(* IEC 61131-3 sources: cc_kush_rewrite/Dumper/POU/Hardware, 4 files *)

(* ---- FB_DumperConveyorMotors.st ---- *)
FUNCTION_BLOCK FB_DumperConveyorMotors
VAR_INPUT
	Dumper : REFERENCE TO ST_Dumper;
	xStart : BOOL;              // Команда запуска
	xStop : BOOL;               // Команда остановки
	xEmergencyStop : BOOL;      // Аварийная остановка
	rTargetFrequency : REAL;    // Целевая частота моторов
END_VAR
VAR_OUTPUT
	eStage : E_StageActuator;   // Текущая стадия
	rCurrentFrequency : REAL;   // Текущая частота моторов (среднее значение)
END_VAR
VAR
	STAGE : E_StageActuator := E_StageActuator.IDLE;

	// Подстадии запуска
	nStartingSubstage : INT := 0;
	// 0 - RELEASE_BRAKE: Отпускание тормоза
	// 1 - WAIT_BRAKE_FEEDBACK: Ожидание обратной связи тормоза
	// 2 - START_VFD: Запуск VFD

	// Подстадии остановки
	nStoppingSubstage : INT := 0;
	// 0 - Нормальная работа
	// 1 - STOP_VFD: Остановка VFD
	// 2 - WAIT_VFD_STOP: Ожидание остановки VFD
	// 3 - ACTIVATE_BRAKE: Активация тормоза
	// 4 - WAIT_BRAKE_FEEDBACK: Ожидание обратной связи тормоза

	// Таймер задержки включения тормоза
	tonTimerEnableBrake : TON;

	// Флаг запуска таймера (защита от зацикливания)
	xBrakeTimerStarted : BOOL := FALSE;
END_VAR

// ========================================
// FB_DumperConveyorMotors - Управление моторами конвейера отвалообразователя
// ========================================
//
// НАЗНАЧЕНИЕ:
// - Управление двумя моторами конвейера (22 кВт каждый)
// - Прямой пуск (без плавного разгона)
// - Последовательная остановка (VFD → тормоз)
// - Не знает про ППЗ и верхнеуровневую логику
// - Просто выполняет команды START/STOP
//
// ВХОДЫ:
// - xStart: команда запуска моторов
// - xStop: команда остановки моторов
// - xEmergencyStop: аварийная остановка
// - rTargetFrequency: целевая частота (Гц)
//
// ВЫХОДЫ:
// - eStage: текущая стадия (IDLE/STARTING/WORK)
// - rCurrentFrequency: текущая частота моторов
//
// ========================================

// ========================================
// ПРИОРИТЕТНАЯ ОБРАБОТКА АВАРИЙНОЙ ОСТАНОВКИ
// ========================================

IF xEmergencyStop THEN
	// Аварийная остановка: немедленное выключение VFD
	Dumper.MotorConveyor[1].VFD.qxStart := FALSE;
	Dumper.MotorConveyor[2].VFD.qxStart := FALSE;

	// Активация тормоза
	Dumper.qxBreakerConveyor := FALSE;

	// Переход в IDLE
	STAGE := E_StageActuator.IDLE;
	nStartingSubstage := 0;
	nStoppingSubstage := 0;
	tonTimerEnableBrake(IN := FALSE);
	xBrakeTimerStarted := FALSE;
END_IF

// ========================================
// АВТОМАТ УПРАВЛЕНИЯ МОТОРАМИ
// ========================================

CASE STAGE OF
	E_StageActuator.IDLE:
		// Сброс подстадий
		nStartingSubstage := 0;
		nStoppingSubstage := 0;

		// Сброс флага таймера тормоза
		xBrakeTimerStarted := FALSE;

		// Тормоз активен (удерживает механизм)
		Dumper.qxBreakerConveyor := FALSE;

		// Команда запуска
		IF xStart AND NOT xEmergencyStop THEN
			STAGE := E_StageActuator.STARTING;
		END_IF

	E_StageActuator.STARTING:
		// Проверка команды остановки во время запуска
		IF xStop THEN
			// Прервать запуск и перейти к остановке
			STAGE := E_StageActuator.WORK;
			nStartingSubstage := 0;
			nStoppingSubstage := 1; // Начать процедуру остановки
		END_IF

		// Последовательный запуск: Тормоз → VFD → Разгон
		CASE nStartingSubstage OF
			0: // RELEASE_BRAKE - Отпускание тормоза
				// Отпустить тормоз (1 = тормоз отпущен)
				Dumper.qxBreakerConveyor := TRUE;

				// Переход к следующей подстадии
				nStartingSubstage := 1;

			1: // WAIT_BRAKE_FEEDBACK - Ожидание обратной связи тормоза
				// Получить обратную связь реле тормоза
				IF Dumper.fbBreakerConveyor.qxSignal THEN
					// Обратная связь получена, переходим к запуску VFD
					nStartingSubstage := 2;
				END_IF

			2: // START_VFD - Запуск VFD
				// Команда ПУСК на частотный преобразователь
				Dumper.MotorConveyor[1].VFD.qxStart := TRUE;
				Dumper.MotorConveyor[2].VFD.qxStart := TRUE;

				// Если оба VFD запущены (обратная связь)
				IF Dumper.MotorConveyor[1].VFD.fbStateIsWorking.qxSignal
					AND Dumper.MotorConveyor[2].VFD.fbStateIsWorking.qxSignal
				THEN
					// Переход в режим WORK
					STAGE := E_StageActuator.WORK;
					nStartingSubstage := 0;
				END_IF
		END_CASE;

	E_StageActuator.WORK:
		// Нормальная работа или штатная остановка через подстадии
		CASE nStoppingSubstage OF
			0: // Нормальная работа
				// Команда остановки
				IF xStop THEN
					nStoppingSubstage := 1;
				END_IF

			1: // STOP_VFD - Остановка VFD
				// Отключить команду пуска на VFD
				Dumper.MotorConveyor[1].VFD.qxStart := FALSE;
				Dumper.MotorConveyor[2].VFD.qxStart := FALSE;

				nStoppingSubstage := 2;

			2: // WAIT_VFD_STOP - Ожидание остановки VFD
				// Проверить обратную связь VFD о выключении
				IF NOT Dumper.MotorConveyor[1].VFD.fbStateIsWorking.qxSignal
					AND NOT Dumper.MotorConveyor[2].VFD.fbStateIsWorking.qxSignal
				THEN
					nStoppingSubstage := 3;
				END_IF

			3: // ACTIVATE_BRAKE - Активация тормоза с задержкой
				// Включение таймера на задержку тормоза (один раз)
				IF NOT xBrakeTimerStarted THEN
					xBrakeTimerStarted := TRUE;
				END_IF

				tonTimerEnableBrake(IN := xBrakeTimerStarted, PT := T#5S);

				IF tonTimerEnableBrake.Q THEN
					// Снять сигнал с тормоза (FALSE = активен)
					Dumper.qxBreakerConveyor := FALSE;
					tonTimerEnableBrake(IN := FALSE);
					xBrakeTimerStarted := FALSE;
					nStoppingSubstage := 4;
				END_IF

			4: // WAIT_BRAKE_FEEDBACK - Переход в IDLE
				STAGE := E_StageActuator.IDLE;
				nStoppingSubstage := 0;
		END_CASE;
END_CASE;

// ========================================
// ЗАДАНИЕ ЧАСТОТЫ МОТОРОВ
// ========================================

// Установка частоты напрямую в аналоговый выход VFD
// В режиме IDLE и при остановке частота = 0
// В режиме WORK частота = rTargetFrequency
IF STAGE = E_StageActuator.WORK THEN
	Dumper.MotorConveyor[1].VFD.qrOutFrequency := rTargetFrequency;
	Dumper.MotorConveyor[2].VFD.qrOutFrequency := rTargetFrequency;
ELSE
	Dumper.MotorConveyor[1].VFD.qrOutFrequency := 0.0;
	Dumper.MotorConveyor[2].VFD.qrOutFrequency := 0.0;
END_IF;

// ========================================
// ВЫХОДЫ
// ========================================

// Текущая стадия
eStage := STAGE;

// Текущая частота (среднее значение двух моторов)
rCurrentFrequency := (Dumper.MotorConveyor[1].VFD.rActualFrequency
                    + Dumper.MotorConveyor[2].VFD.rActualFrequency) / 2.0;

END_FUNCTION_BLOCK

(* ---- FB_DumperMotorErrors.st ---- *)
FUNCTION_BLOCK FB_DumperMotorErrors
VAR_INPUT
	Dumper : REFERENCE TO ST_Dumper;
END_VAR
VAR_OUTPUT
	// Ошибки моторов конвейера
	xErrorMotorConv1 : BOOL;
	xErrorMotorConv2 : BOOL;
	xErrorMotorConv_Any : BOOL;

	// Ошибки моторов поворота
	xErrorMotorRot1 : BOOL;
	xErrorMotorRot2 : BOOL;
	xErrorMotorRot_Any : BOOL;

	// Агрегированный выход
	xErrorMotors : BOOL; // Любая ошибка моторов
END_VAR

// ========================================
// FB_DumperMotorErrors - Проверка ошибок моторов отвалообразователя
// ========================================
//
// НАЗНАЧЕНИЕ:
// - Проверка всех моторов отвалообразователя на ошибки
// - Формирование индивидуальных флагов ошибок
// - Агрегирование ошибок
//
// МОТОРЫ:
// - MotorConveyor[1..2]: Моторы конвейера (22 кВт)
// - MotorRotation[1..2]: Моторы поворота (3 кВт)
//
// ПРОВЕРЯЕМЫЕ ОШИБКИ:
// - Ошибка VFD (fbStateFailure: 0 = ошибка, 1 = норма, NC контакт)
//
// ========================================

// ========================================
// ПРОВЕРКА МОТОРОВ КОНВЕЙЕРА
// ========================================

// Мотор конвейера 1
// fbStateFailure - NC контакт: 0 = ошибка VFD, 1 = норма
xErrorMotorConv1 := NOT Dumper.MotorConveyor[1].VFD.fbStateFailure.qxSignal;

// Мотор конвейера 2
xErrorMotorConv2 := NOT Dumper.MotorConveyor[2].VFD.fbStateFailure.qxSignal;

xErrorMotorConv_Any := xErrorMotorConv1 OR xErrorMotorConv2;

// ========================================
// ПРОВЕРКА МОТОРОВ ПОВОРОТА
// ========================================

// Мотор поворота 1
xErrorMotorRot1 := NOT Dumper.MotorRotation[1].VFD.fbStateFailure.qxSignal;

// Мотор поворота 2
xErrorMotorRot2 := NOT Dumper.MotorRotation[2].VFD.fbStateFailure.qxSignal;

xErrorMotorRot_Any := xErrorMotorRot1 OR xErrorMotorRot2;

// ========================================
// АГРЕГИРОВАНИЕ ОШИБОК
// ========================================

xErrorMotors := xErrorMotorConv_Any OR xErrorMotorRot_Any;

END_FUNCTION_BLOCK

(* ---- FB_DumperRotationMotors.st ---- *)
FUNCTION_BLOCK FB_DumperRotationMotors
VAR_INPUT
	Dumper : REFERENCE TO ST_Dumper;
	xTurnLeft : BOOL;           // Команда поворота влево
	xTurnRight : BOOL;          // Команда поворота вправо
	xStop : BOOL;               // Команда остановки поворота
	xEmergencyStop : BOOL;      // Аварийная остановка
	rTargetFrequency : REAL;    // Целевая частота моторов
END_VAR
VAR_OUTPUT
	eStage : E_StageActuator;   // Текущая стадия
	rCurrentFrequency : REAL;   // Текущая частота моторов (среднее значение)
	xRotatingLeft : BOOL;       // Активен поворот влево
	xRotatingRight : BOOL;      // Активен поворот вправо
END_VAR
VAR
	STAGE : E_StageActuator := E_StageActuator.IDLE;

	// Направление поворота
	xLeftActive : BOOL := FALSE;  // Поворот влево активен
	xRightActive : BOOL := FALSE; // Поворот вправо активен

	// Подстадии запуска
	nStartingSubstage : INT := 0;
	// 0 - IDLE
	// 1 - RELEASE_BRAKE: Отпускание тормоза поворота
	// 2 - WAIT_BRAKE_FEEDBACK: Ожидание обратной связи тормоза
	// 3 - START_VFD: Запуск VFD поворота

	// Подстадии остановки
	nStoppingSubstage : INT := 0;
	// 0 - Нормальная работа
	// 1 - STOP_VFD: Остановка VFD
	// 2 - WAIT_VFD_STOP: Ожидание остановки VFD
	// 3 - ACTIVATE_BRAKE: Активация тормоза

	// Таймер задержки включения тормоза
	tonTimerEnableBrake : TON;

	// Флаг запуска таймера (защита от зацикливания)
	xBrakeTimerStarted : BOOL := FALSE;
END_VAR

// ========================================
// FB_DumperRotationMotors - Управление моторами поворота отвалообразователя
// ========================================
//
// НАЗНАЧЕНИЕ:
// - Управление двумя моторами поворота (3 кВт каждый)
// - Поддержка реверса (влево/вправо)
// - Блокировка по концевым выключателям
// - Последовательная остановка (VFD → тормоз)
// - Не знает про верхнеуровневую логику
// - Просто выполняет команды TURN_LEFT/TURN_RIGHT/STOP
//
// ВХОДЫ:
// - xTurnLeft: команда поворота влево
// - xTurnRight: команда поворота вправо
// - xStop: команда остановки
// - xEmergencyStop: аварийная остановка
// - rTargetFrequency: целевая частота (Гц)
//
// ВЫХОДЫ:
// - eStage: текущая стадия (IDLE/STARTING/WORK)
// - rCurrentFrequency: текущая частота моторов
// - xRotatingLeft: флаг активного поворота влево
// - xRotatingRight: флаг активного поворота вправо
//
// ========================================

// ========================================
// ПРИОРИТЕТНАЯ ОБРАБОТКА АВАРИЙНОЙ ОСТАНОВКИ
// ========================================

IF xEmergencyStop THEN
	// Аварийная остановка: немедленное выключение VFD
	Dumper.MotorRotation[1].VFD.qxStart := FALSE;
	Dumper.MotorRotation[2].VFD.qxStart := FALSE;
	Dumper.MotorRotation[1].qxVFDReverseStart := FALSE;
	Dumper.MotorRotation[2].qxVFDReverseStart := FALSE;

	// Активация тормоза
	Dumper.qxBreakerRotation := FALSE;

	// Сброс направления
	xLeftActive := FALSE;
	xRightActive := FALSE;

	// Переход в IDLE
	STAGE := E_StageActuator.IDLE;
	nStartingSubstage := 0;
	nStoppingSubstage := 0;
	tonTimerEnableBrake(IN := FALSE);
	xBrakeTimerStarted := FALSE;
END_IF

// ========================================
// АВТОМАТ УПРАВЛЕНИЯ МОТОРАМИ ПОВОРОТА
// ========================================

CASE STAGE OF
	E_StageActuator.IDLE:
		// Сброс подстадий
		nStartingSubstage := 0;
		nStoppingSubstage := 0;

		// Сброс флага таймера тормоза
		xBrakeTimerStarted := FALSE;

		// Тормоз активен
		Dumper.qxBreakerRotation := FALSE;

		// Остановка VFD
		Dumper.MotorRotation[1].VFD.qxStart := FALSE;
		Dumper.MotorRotation[2].VFD.qxStart := FALSE;
		Dumper.MotorRotation[1].qxVFDReverseStart := FALSE;
		Dumper.MotorRotation[2].qxVFDReverseStart := FALSE;

		// Сброс флагов направления
		xLeftActive := FALSE;
		xRightActive := FALSE;

		// Команда поворота влево
		IF xTurnLeft AND NOT xEmergencyStop AND NOT xTurnRight THEN
			// Проверка концевого выключателя влево
			// qxSignal = TRUE означает концевик в норме (не нажат)
			IF Dumper.fbEndSwitchLeft.qxSignal THEN
				xLeftActive := TRUE;
				xRightActive := FALSE;
				STAGE := E_StageActuator.STARTING;
			END_IF
		END_IF

		// Команда поворота вправо
		IF xTurnRight AND NOT xEmergencyStop AND NOT xTurnLeft THEN
			// Проверка концевого выключателя вправо
			IF Dumper.fbEndSwitchRight.qxSignal THEN
				xRightActive := TRUE;
				xLeftActive := FALSE;
				STAGE := E_StageActuator.STARTING;
			END_IF
		END_IF

	E_StageActuator.STARTING:
		// Проверка команды остановки во время запуска
		IF xStop THEN
			// Прервать запуск и перейти к остановке
			STAGE := E_StageActuator.WORK;
			nStartingSubstage := 0;
			nStoppingSubstage := 1; // Начать процедуру остановки
		END_IF

		// Проверка достижения концевого выключателя
		IF (xLeftActive AND NOT Dumper.fbEndSwitchLeft.qxSignal)
			OR (xRightActive AND NOT Dumper.fbEndSwitchRight.qxSignal)
		THEN
			// Концевик достигнут, начать остановку
			STAGE := E_StageActuator.WORK;
			nStartingSubstage := 0;
			nStoppingSubstage := 1;
		END_IF

		// Последовательный запуск: Тормоз → VFD → Разгон
		CASE nStartingSubstage OF
			0: // IDLE
				nStartingSubstage := 1;

			1: // RELEASE_BRAKE - Отпускание тормоза
				// Отпустить тормоз (1 = тормоз отпущен)
				Dumper.qxBreakerRotation := TRUE;

				// Переход к следующей подстадии
				nStartingSubstage := 2;

			2: // WAIT_BRAKE_FEEDBACK - Ожидание обратной связи тормоза
				// Получить обратную связь реле тормоза
				IF Dumper.fbBreakerRotation.qxSignal THEN
					// Обратная связь получена, переходим к запуску VFD
					nStartingSubstage := 3;
				END_IF

			3: // START_VFD - Запуск VFD
				// Установка направления и запуск VFD
				IF xLeftActive THEN
					// Поворот влево - прямое направление
					Dumper.MotorRotation[1].qxVFDReverseStart := FALSE;
					Dumper.MotorRotation[2].qxVFDReverseStart := FALSE;
					Dumper.MotorRotation[1].VFD.qxStart := TRUE;
					Dumper.MotorRotation[2].VFD.qxStart := TRUE;
				ELSIF xRightActive THEN
					// Поворот вправо - реверс
					Dumper.MotorRotation[1].VFD.qxStart := FALSE;
					Dumper.MotorRotation[2].VFD.qxStart := FALSE;
					Dumper.MotorRotation[1].qxVFDReverseStart := TRUE;
					Dumper.MotorRotation[2].qxVFDReverseStart := TRUE;
				END_IF

				// Проверка запуска VFD (обратная связь)
				IF Dumper.MotorRotation[1].VFD.fbStateIsWorking.qxSignal
					AND Dumper.MotorRotation[2].VFD.fbStateIsWorking.qxSignal
				THEN
					// VFD запущены, переходим в режим работы
					STAGE := E_StageActuator.WORK;
					nStartingSubstage := 0;
				END_IF
		END_CASE;

	E_StageActuator.WORK:
		// Нормальная работа или штатная остановка через подстадии
		CASE nStoppingSubstage OF
			0: // Нормальная работа
				// Проверка команды остановки
				IF xStop THEN
					nStoppingSubstage := 1;
				END_IF

				// Проверка достижения концевого выключателя
				IF (xLeftActive AND NOT Dumper.fbEndSwitchLeft.qxSignal)
					OR (xRightActive AND NOT Dumper.fbEndSwitchRight.qxSignal)
				THEN
					// Концевик достигнут, автоматическая остановка
					nStoppingSubstage := 1;
				END_IF

			1: // STOP_VFD - Остановка VFD
				// Отключить команду пуска на VFD
				Dumper.MotorRotation[1].VFD.qxStart := FALSE;
				Dumper.MotorRotation[2].VFD.qxStart := FALSE;
				Dumper.MotorRotation[1].qxVFDReverseStart := FALSE;
				Dumper.MotorRotation[2].qxVFDReverseStart := FALSE;

				nStoppingSubstage := 2;

			2: // WAIT_VFD_STOP - Ожидание остановки VFD
				// Проверить обратную связь VFD о выключении
				IF NOT Dumper.MotorRotation[1].VFD.fbStateIsWorking.qxSignal
					AND NOT Dumper.MotorRotation[2].VFD.fbStateIsWorking.qxSignal
				THEN
					nStoppingSubstage := 3;
				END_IF

			3: // ACTIVATE_BRAKE - Активация тормоза с задержкой
				// Включение таймера на задержку тормоза (один раз)
				IF NOT xBrakeTimerStarted THEN
					xBrakeTimerStarted := TRUE;
				END_IF

				tonTimerEnableBrake(IN := xBrakeTimerStarted, PT := T#3S);

				IF tonTimerEnableBrake.Q THEN
					// Снять сигнал с тормоза (FALSE = активен)
					Dumper.qxBreakerRotation := FALSE;
					tonTimerEnableBrake(IN := FALSE);
					xBrakeTimerStarted := FALSE;

					// Сброс флагов направления
					xLeftActive := FALSE;
					xRightActive := FALSE;

					// Переход в IDLE
					STAGE := E_StageActuator.IDLE;
					nStoppingSubstage := 0;
				END_IF
		END_CASE;
END_CASE;

// ========================================
// ЗАДАНИЕ ЧАСТОТЫ МОТОРОВ
// ========================================

// Установка частоты напрямую в аналоговый выход VFD
// В режиме IDLE и при остановке частота = 0
// В режиме WORK частота = rTargetFrequency
IF STAGE = E_StageActuator.WORK THEN
	Dumper.MotorRotation[1].VFD.qrOutFrequency := rTargetFrequency;
	Dumper.MotorRotation[2].VFD.qrOutFrequency := rTargetFrequency;
ELSE
	Dumper.MotorRotation[1].VFD.qrOutFrequency := 0.0;
	Dumper.MotorRotation[2].VFD.qrOutFrequency := 0.0;
END_IF;

// ========================================
// ВЫХОДЫ
// ========================================

// Текущая стадия
eStage := STAGE;

// Текущая частота (среднее значение двух моторов)
rCurrentFrequency := (Dumper.MotorRotation[1].VFD.rActualFrequency
                    + Dumper.MotorRotation[2].VFD.rActualFrequency) / 2.0;

// Флаги активного поворота
xRotatingLeft := xLeftActive;
xRotatingRight := xRightActive;

END_FUNCTION_BLOCK

(* ---- FB_DumperSensors.st ---- *)
FUNCTION_BLOCK FB_DumperSensors
VAR_INPUT
	Dumper : REFERENCE TO ST_Dumper;
	xReset : BOOL; // Команда сброса зафиксированных ошибок
END_VAR
VAR_OUTPUT
	// Ошибки по датчикам схода ленты (ZQ Alarm)
	xErrorZQ1 : BOOL;
	xErrorZQ2 : BOOL;
	xErrorZQ3 : BOOL;
	xErrorZQ4 : BOOL;
	xErrorZQ_Any : BOOL; // Любая ошибка ZQ

	// Предупреждения по датчикам схода ленты (ZQ Warning)
	xWarningZQ1 : BOOL;
	xWarningZQ2 : BOOL;
	xWarningZQ3 : BOOL;
	xWarningZQ4 : BOOL;
	xWarningZQ_Any : BOOL; // Любое предупреждение ZQ

	// Ошибки по кабель-тросовым выключателям (HQ)
	xErrorHQ1 : BOOL;
	xErrorHQ2 : BOOL;
	xErrorHQ3 : BOOL;
	xErrorHQ4 : BOOL;
	xErrorHQ_Any : BOOL; // Любая ошибка HQ

	// Ошибки по ограждениям барабана (SQ)
	xErrorSQ1 : BOOL;
	xErrorSQ2 : BOOL;
	xErrorSQ_Any : BOOL; // Любая ошибка SQ

	// Ошибка контроля заштыбовки (GS)
	xErrorGS : BOOL;

	// Ошибки датчиков скорости (QR)
	xErrorQR1 : BOOL;
	xErrorQR2 : BOOL;
	xErrorQR_Any : BOOL; // Любая ошибка QR

	// Ошибка контроля продольного разрыва (YS)
	xErrorYS : BOOL;

	// Агрегированные выходы
	xErrorSafetySensors : BOOL;  // Любая ошибка датчиков безопасности
	xWarningSafetySensors : BOOL; // Любое предупреждение датчиков безопасности
END_VAR
VAR
	// Внутренние переменные для фиксации ошибок (текущие состояния без фиксации)
	_xCurrentErrorZQ1 : BOOL;
	_xCurrentErrorZQ2 : BOOL;
	_xCurrentErrorZQ3 : BOOL;
	_xCurrentErrorZQ4 : BOOL;

	_xCurrentWarningZQ1 : BOOL;
	_xCurrentWarningZQ2 : BOOL;
	_xCurrentWarningZQ3 : BOOL;
	_xCurrentWarningZQ4 : BOOL;

	_xCurrentErrorHQ1 : BOOL;
	_xCurrentErrorHQ2 : BOOL;
	_xCurrentErrorHQ3 : BOOL;
	_xCurrentErrorHQ4 : BOOL;

	_xCurrentErrorSQ1 : BOOL;
	_xCurrentErrorSQ2 : BOOL;

	_xCurrentErrorGS : BOOL;
	_xCurrentErrorQR1 : BOOL;
	_xCurrentErrorQR2 : BOOL;
	_xCurrentErrorYS : BOOL;

	// RS-триггеры для фиксации ошибок
	_fbLatchErrorZQ1 : RS;
	_fbLatchErrorZQ2 : RS;
	_fbLatchErrorZQ3 : RS;
	_fbLatchErrorZQ4 : RS;

	_fbLatchWarningZQ1 : RS;
	_fbLatchWarningZQ2 : RS;
	_fbLatchWarningZQ3 : RS;
	_fbLatchWarningZQ4 : RS;

	_fbLatchErrorHQ1 : RS;
	_fbLatchErrorHQ2 : RS;
	_fbLatchErrorHQ3 : RS;
	_fbLatchErrorHQ4 : RS;

	_fbLatchErrorSQ1 : RS;
	_fbLatchErrorSQ2 : RS;

	_fbLatchErrorGS : RS;
	_fbLatchErrorQR1 : RS;
	_fbLatchErrorQR2 : RS;
	_fbLatchErrorYS : RS;
END_VAR

// ========================================
// FB_DumperSensors - Обработка датчиков безопасности отвалообразователя
// ========================================
//
// НАЗНАЧЕНИЕ:
// - Мониторинг всех датчиков безопасности
// - Фиксация ошибок через RS-триггеры (память до сброса)
// - Формирование индивидуальных флагов ошибок
// - Агрегирование ошибок и предупреждений
//
// ДАТЧИКИ:
// - ZQ (1-4): Контроль схода ленты (Alarm + Warning)
// - HQ (1-4): Кабель-тросовый выключатель (аварийная остановка)
// - SQ (1-2): Контроль ограждения барабана
// - GS: Контроль заштыбовки
// - QR (1-2): Измерение скорости вращения барабана
// - YS: Контроль продольного разрыва ленты
//
// ЛОГИКА ФИКСАЦИИ:
// - При возникновении ошибки она фиксируется (SET в RS-триггер)
// - Ошибка сохраняется даже после устранения неисправности датчика
// - Сброс всех зафиксированных ошибок через вход xReset
//
// ВЫХОДЫ:
// - Индивидуальные флаги для каждого датчика (зафиксированные)
// - Агрегированные флаги (Any) для групп датчиков
// - Общие флаги ошибок и предупреждений
//
// ========================================

// ========================================
// ДАТЧИКИ СХОДА ЛЕНТЫ (ZQ) - ALARM
// ========================================
// Логика: 1 = Норма, 0 = Тревога (сход ленты)

// Определяем текущее состояние датчиков
_xCurrentErrorZQ1 := NOT Dumper.fbZQAlarm[1].qxSignal;
_xCurrentErrorZQ2 := NOT Dumper.fbZQAlarm[2].qxSignal;
_xCurrentErrorZQ3 := NOT Dumper.fbZQAlarm[3].qxSignal;
_xCurrentErrorZQ4 := NOT Dumper.fbZQAlarm[4].qxSignal;

// Фиксируем ошибки через RS-триггеры (SET при ошибке, RESET по команде xReset)
_fbLatchErrorZQ1(SET := _xCurrentErrorZQ1, RESET1 := xReset);
_fbLatchErrorZQ2(SET := _xCurrentErrorZQ2, RESET1 := xReset);
_fbLatchErrorZQ3(SET := _xCurrentErrorZQ3, RESET1 := xReset);
_fbLatchErrorZQ4(SET := _xCurrentErrorZQ4, RESET1 := xReset);

// Выходы - зафиксированные ошибки
xErrorZQ1 := _fbLatchErrorZQ1.Q1;
xErrorZQ2 := _fbLatchErrorZQ2.Q1;
xErrorZQ3 := _fbLatchErrorZQ3.Q1;
xErrorZQ4 := _fbLatchErrorZQ4.Q1;

xErrorZQ_Any := xErrorZQ1 OR xErrorZQ2 OR xErrorZQ3 OR xErrorZQ4;

// ========================================
// ДАТЧИКИ СХОДА ЛЕНТЫ (ZQ) - WARNING
// ========================================
// Логика: 1 = Норма, 0 = Предупреждение (лента близка к сходу)

// Определяем текущее состояние датчиков
_xCurrentWarningZQ1 := NOT Dumper.fbZQWarning[1].qxSignal;
_xCurrentWarningZQ2 := NOT Dumper.fbZQWarning[2].qxSignal;
_xCurrentWarningZQ3 := NOT Dumper.fbZQWarning[3].qxSignal;
_xCurrentWarningZQ4 := NOT Dumper.fbZQWarning[4].qxSignal;

// Фиксируем предупреждения через RS-триггеры
_fbLatchWarningZQ1(SET := _xCurrentWarningZQ1, RESET1 := xReset);
_fbLatchWarningZQ2(SET := _xCurrentWarningZQ2, RESET1 := xReset);
_fbLatchWarningZQ3(SET := _xCurrentWarningZQ3, RESET1 := xReset);
_fbLatchWarningZQ4(SET := _xCurrentWarningZQ4, RESET1 := xReset);

// Выходы - зафиксированные предупреждения
xWarningZQ1 := _fbLatchWarningZQ1.Q1;
xWarningZQ2 := _fbLatchWarningZQ2.Q1;
xWarningZQ3 := _fbLatchWarningZQ3.Q1;
xWarningZQ4 := _fbLatchWarningZQ4.Q1;

xWarningZQ_Any := xWarningZQ1 OR xWarningZQ2 OR xWarningZQ3 OR xWarningZQ4;

// ========================================
// КАБЕЛЬ-ТРОСОВЫЕ ВЫКЛЮЧАТЕЛИ (HQ)
// ========================================
// Логика: 1 = Норма, 0 = Аварийная остановка (трос натянут)

// Определяем текущее состояние датчиков
_xCurrentErrorHQ1 := NOT Dumper.fbHQ_IsOk[1].qxSignal;
_xCurrentErrorHQ2 := NOT Dumper.fbHQ_IsOk[2].qxSignal;
_xCurrentErrorHQ3 := NOT Dumper.fbHQ_IsOk[3].qxSignal;
_xCurrentErrorHQ4 := NOT Dumper.fbHQ_IsOk[4].qxSignal;

// Фиксируем ошибки через RS-триггеры
_fbLatchErrorHQ1(SET := _xCurrentErrorHQ1, RESET1 := xReset);
_fbLatchErrorHQ2(SET := _xCurrentErrorHQ2, RESET1 := xReset);
_fbLatchErrorHQ3(SET := _xCurrentErrorHQ3, RESET1 := xReset);
_fbLatchErrorHQ4(SET := _xCurrentErrorHQ4, RESET1 := xReset);

// Выходы - зафиксированные ошибки
xErrorHQ1 := _fbLatchErrorHQ1.Q1;
xErrorHQ2 := _fbLatchErrorHQ2.Q1;
xErrorHQ3 := _fbLatchErrorHQ3.Q1;
xErrorHQ4 := _fbLatchErrorHQ4.Q1;

xErrorHQ_Any := xErrorHQ1 OR xErrorHQ2 OR xErrorHQ3 OR xErrorHQ4;

// ========================================
// КОНТРОЛЬ ОГРАЖДЕНИЯ БАРАБАНА (SQ)
// ========================================
// Логика: 1 = Норма (ограждение закрыто), 0 = Тревога (ограждение открыто)

// Определяем текущее состояние датчиков
_xCurrentErrorSQ1 := NOT Dumper.fbSQ_IsOk[1].qxSignal;
_xCurrentErrorSQ2 := NOT Dumper.fbSQ_IsOk[2].qxSignal;

// Фиксируем ошибки через RS-триггеры
_fbLatchErrorSQ1(SET := _xCurrentErrorSQ1, RESET1 := xReset);
_fbLatchErrorSQ2(SET := _xCurrentErrorSQ2, RESET1 := xReset);

// Выходы - зафиксированные ошибки
xErrorSQ1 := _fbLatchErrorSQ1.Q1;
xErrorSQ2 := _fbLatchErrorSQ2.Q1;

xErrorSQ_Any := xErrorSQ1 OR xErrorSQ2;

// ========================================
// КОНТРОЛЬ ЗАШТЫБОВКИ (GS)
// ========================================
// Логика: 1 = Норма, 0 = Тревога (заштыбовка материала)

// Определяем текущее состояние датчика
_xCurrentErrorGS := NOT Dumper.fbGS1.qxSignal;

// Фиксируем ошибку через RS-триггер
_fbLatchErrorGS(SET := _xCurrentErrorGS, RESET1 := xReset);

// Выход - зафиксированная ошибка
xErrorGS := _fbLatchErrorGS.Q1;

// ========================================
// ДАТЧИКИ СКОРОСТИ (QR)
// ========================================
// Логика: Проверка наличия импульсов (детектирование остановки при работающем моторе)
// Ошибка определяется на верхнем уровне по сравнению с состоянием мотора

// Определяем текущее состояние датчиков (резерв для будущей реализации)
_xCurrentErrorQR1 := FALSE; // Резерв для будущей реализации
_xCurrentErrorQR2 := FALSE; // Резерв для будущей реализации

// Фиксируем ошибки через RS-триггеры
_fbLatchErrorQR1(SET := _xCurrentErrorQR1, RESET1 := xReset);
_fbLatchErrorQR2(SET := _xCurrentErrorQR2, RESET1 := xReset);

// Выходы - зафиксированные ошибки
xErrorQR1 := _fbLatchErrorQR1.Q1;
xErrorQR2 := _fbLatchErrorQR2.Q1;

xErrorQR_Any := xErrorQR1 OR xErrorQR2;

// ========================================
// КОНТРОЛЬ ПРОДОЛЬНОГО РАЗРЫВА (YS)
// ========================================
// Логика: 1 = Норма, 0 = Тревога (продольный разрыв ленты)

// Определяем текущее состояние датчика
_xCurrentErrorYS := NOT Dumper.fbYS1.qxSignal;

// Фиксируем ошибку через RS-триггер
_fbLatchErrorYS(SET := _xCurrentErrorYS, RESET1 := xReset);

// Выход - зафиксированная ошибка
xErrorYS := _fbLatchErrorYS.Q1;

// ========================================
// АГРЕГИРОВАНИЕ ОШИБОК И ПРЕДУПРЕЖДЕНИЙ
// ========================================

// Все критические ошибки датчиков безопасности
xErrorSafetySensors := xErrorZQ_Any    // Сход ленты (критический уровень)
                    OR xErrorHQ_Any     // Аварийная остановка по тросу
                    OR xErrorSQ_Any     // Открыто ограждение
                    OR xErrorGS         // Заштыбовка
                    OR xErrorQR_Any     // Остановка барабана
                    OR xErrorYS;        // Продольный разрыв

// Все предупреждения датчиков безопасности
xWarningSafetySensors := xWarningZQ_Any; // Предупреждение схода ленты

END_FUNCTION_BLOCK
